TYPE Verbruik_input :
STRUCT
	Puls		AT %I*	: BOOL;
	Value				: REAL;
//	Meetgegevens		: ST_Meetgegevens;
END_STRUCT
END_TYPE

(* stored: Version 1.1.0.1, ProductVersion 3.1.4024.12
   DUT Verbruik_input: Id {a05d517b-4a45-4c4c-8488-b25b2e378fab} *)
